(* Logix 5000 project; controller STAT 1756-L72 rev 20.12; software revision 20.04; part 8 of 34 *)
(* tags used below, declared in another part *)
   B14 : DINT[30];
   B3 : DINT[256];
   dmd_soude_ibt_ok : BOOL;
   FRANCK : BOOL;
   I10_000_Bit07 : ALIAS FOR I10[0].7;   // Hand Automaat CL8
   I10_001_Bit07 : ALIAS FOR I10[1].7;   // Hand Automaat CL9
   I19_000_Bit09 : ALIAS FOR I19[0].9;   // BP RESET KLAXON
   I1_008_Bit01 : ALIAS FOR I1[8].1;   // Hand Automaat stormbekken
   I8_001_Bit01 : ALIAS FOR I8[1].1;   // hand automaat cl5
   I8_001_Bit09 : ALIAS FOR I8[1].9;   // Schakelaar hand autom cl6
   I9_000_Bit09 : ALIAS FOR I9[0].9;   // Hand_Auto CL7
   ibt_level_soude_plein : BOOL;
   N12 : DINT[230];
   O12_000_Bit00 : ALIAS FOR O12[0].0;   // spoelpomp filters dubbele media P6_SPOEL
   O12_000_Bit01 : ALIAS FOR O12[0].1;   // pomp pompen uit kelder P23_KELDER
   O12_000_Bit02 : ALIAS FOR O12[0].2;   // pomp pompen uit kelder P24_KELDER
   O12_000_Bit03 : ALIAS FOR O12[0].3;   // motor ag1 mixer krimp neutralisatie AG1_MIXER_KRIMP
   O12_000_Bit08 : ALIAS FOR O12[0].8;   // pomp ag2 mixer vat 1 AG2_MIXER_VAT1
   O12_000_Bit09 : ALIAS FOR O12[0].9;   // pomp ag3 mixer vat 2 AG3_MIXER_VAT2
   O12_000_Bit10 : ALIAS FOR O12[0].10;   // pomp pd7 doseerpomp floculaat PD7_DOSEER_FLOCU
   O12_000_Bit11 : ALIAS FOR O12[0].11;   // pomp pd8 doseerpomp floculaat PD8_DOSEER_FLOCU
   O12_000_Bit12 : ALIAS FOR O12[0].12;   // Motor P19a zuiveringspomp controleweger P19_ZUIVERP
   O12_000_Bit13 : ALIAS FOR O12[0].13;   // Motor P20 zuiveringspomp controleweger P20_ZUIVERP
   O12_000_Bit14 : ALIAS FOR O12[0].14;   // Motor Pm1 recerculatiepomp ingang 1 decanter PM1_RECER_DEC1
   O12_000_Bit15 : ALIAS FOR O12[0].15;   // Motor Pm2 recerculatiepomp ingang 2 decanter PM2_RECER_DEC2
   O12_001_Bit00 : ALIAS FOR O12[1].0;   // Motor Pm3 evacuatiepomp ingang 1 decanter PM3_EVACU_IN_1
   O12_001_Bit01 : ALIAS FOR O12[1].1;   // Motor Pm4 evacuatiepomp ingang 2 decanter PM4_EVACU_IN_2
   O12_001_Bit03 : ALIAS FOR O12[1].3;   // Motor P7 voedingspomp omgekeerde osmose 1 P7_OSMOSE_1
   O12_001_Bit04 : ALIAS FOR O12[1].4;   // Motor P8 voedingspomp omgekeerde osmose 2 P8_OSMOSE_2
   O12_001_Bit05 : ALIAS FOR O12[1].5;   // Motor P9 voedingspomp omgekeerde osmose 3 P9_OSMOSE_3
   O14_001_Bit04 : ALIAS FOR O14[1].4;   // kalxon out NAOH
   O14_001_Bit05 : ALIAS FOR O14[1].5;   // lampe out NAOH
   O14_001_Bit06 : ALIAS FOR O14[1].6;   // klaxon out H2SO4
   O14_001_Bit07 : ALIAS FOR O14[1].7;   // lampe H2SO4
   O14_001_Bit08 : ALIAS FOR O14[1].8;   // klaxon out ZOUT
   O14_001_Bit09 : ALIAS FOR O14[1].9;   // lampe ZOUT
   O16_000_Bit09 : ALIAS FOR O16[0].9;   // LAMP_P17_AAN
   O16_000_Bit10 : ALIAS FOR O16[0].10;   // LAMP_P17_UIT
   O16_000_Bit11 : ALIAS FOR O16[0].11;   // LAMP_P18_AAN
   O16_000_Bit12 : ALIAS FOR O16[0].12;   // LAMP_P18_UIT
   O16_000_Bit15 : ALIAS FOR O16[0].15;   // LAMP_PRO1_AAN
   O16_001_Bit00 : ALIAS FOR O16[1].0;   // LAMP_PRO1_UIT
   O16_001_Bit01 : ALIAS FOR O16[1].1;   // LAMP_PRO2_AAN
   O16_001_Bit02 : ALIAS FOR O16[1].2;   // LAMP_PRO2_UIT
   O16_001_Bit03 : ALIAS FOR O16[1].3;   // LAMP_P21_AAN
   O16_001_Bit04 : ALIAS FOR O16[1].4;   // LAMP_P21_UIT
   O16_001_Bit05 : ALIAS FOR O16[1].5;   // LAMP_P22_AAN
   O16_001_Bit06 : ALIAS FOR O16[1].6;   // LAMP_P22_UIT
   O16_001_Bit07 : ALIAS FOR O16[1].7;   // LAMP_PRO3_AAN
   O16_001_Bit08 : ALIAS FOR O16[1].8;   // LAMP_PRO3_UIT
   O16_001_Bit09 : ALIAS FOR O16[1].9;   // LAMP_P21_REINIG_AAN
   O16_001_Bit10 : ALIAS FOR O16[1].10;   // LAMP_P21_REINIG_UIT
   O16_001_Bit11 : ALIAS FOR O16[1].11;   // LAMP_VENT_S1_AAN
   O16_001_Bit12 : ALIAS FOR O16[1].12;   // LAMP_VENT_S1_UIT
   O16_001_Bit13 : ALIAS FOR O16[1].13;   // LAMP_P3_AAN
   O16_001_Bit14 : ALIAS FOR O16[1].14;   // LAMP_P3_UIT
   O16_001_Bit15 : ALIAS FOR O16[1].15;   // LAMP_P4_AAN
   O17_000_Bit00 : ALIAS FOR O17[0].0;   // LAMP_P4_UIT
   O17_000_Bit01 : ALIAS FOR O17[0].1;   // LAMP_P5_AAN
   O17_000_Bit02 : ALIAS FOR O17[0].2;   // LAMP_P5_UIT
   O17_000_Bit03 : ALIAS FOR O17[0].3;   // LAMP_P6_AAN
   O17_000_Bit04 : ALIAS FOR O17[0].4;   // LAMP_P6_UIT
   O17_000_Bit05 : ALIAS FOR O17[0].5;   // LAMP_P23_AAN
   O17_000_Bit06 : ALIAS FOR O17[0].6;   // LAMP_P23_UIT
   O17_000_Bit07 : ALIAS FOR O17[0].7;   // LAMP_P24_AAN
   O17_000_Bit08 : ALIAS FOR O17[0].8;   // LAMP_P24_UIT
   O17_000_Bit09 : ALIAS FOR O17[0].9;   // LAMP_AG1_AAN
   O17_000_Bit10 : ALIAS FOR O17[0].10;   // LAMP_AG1_UIT
   O17_000_Bit11 : ALIAS FOR O17[0].11;   // LAMP_AG2_AAN
   O17_000_Bit12 : ALIAS FOR O17[0].12;   // LAMP_AG2_UIT
   O17_000_Bit13 : ALIAS FOR O17[0].13;   // LAMP_AG3_AAN
   O17_000_Bit14 : ALIAS FOR O17[0].14;   // LAMP_AG3_UIT
   O17_000_Bit15 : ALIAS FOR O17[0].15;   // LAMP_PD7_AAN
   O17_001_Bit00 : ALIAS FOR O17[1].0;   // LAMP_PD7_UIT
   O17_001_Bit01 : ALIAS FOR O17[1].1;   // LAMP_PD8_AAN
   O17_001_Bit02 : ALIAS FOR O17[1].2;   // LAMP_PD8_UIT
   O17_001_Bit03 : ALIAS FOR O17[1].3;   // LAMP_P19A_AAN
   O17_001_Bit04 : ALIAS FOR O17[1].4;   // LAMP_P19A_UIT
   O17_001_Bit05 : ALIAS FOR O17[1].5;   // LAMP_P19B_AAN
   O17_001_Bit06 : ALIAS FOR O17[1].6;   // LAMP_P19B_UIT
   O17_001_Bit09 : ALIAS FOR O17[1].9;   // LAMP_P25_AAN
   O17_001_Bit10 : ALIAS FOR O17[1].10;   // LAMP_P25_UIT
   O17_001_Bit11 : ALIAS FOR O17[1].11;   // LAMP_PM1_AAN
   O17_001_Bit12 : ALIAS FOR O17[1].12;   // LAMP_PM1_UIT
   O17_001_Bit13 : ALIAS FOR O17[1].13;   // LAMP_PM2_AAN
   O17_001_Bit14 : ALIAS FOR O17[1].14;   // LAMP_PM2_UIT
   O17_001_Bit15 : ALIAS FOR O17[1].15;   // LAMP_PM3_AAN
   O18_000_Bit00 : ALIAS FOR O18[0].0;   // LAMP_PM3_UIT
   O18_000_Bit01 : ALIAS FOR O18[0].1;   // LAMP_PM4_AAN
   O18_000_Bit02 : ALIAS FOR O18[0].2;   // LAMP_PM4_UIT
   O18_000_Bit07 : ALIAS FOR O18[0].7;   // LAMP_P7_AAN
   O18_000_Bit08 : ALIAS FOR O18[0].8;   // LAMP_P7_UIT
   O18_000_Bit09 : ALIAS FOR O18[0].9;   // LAMP_P8_AAN
   O18_000_Bit10 : ALIAS FOR O18[0].10;   // LAMP_P8_UIT
   O18_000_Bit11 : ALIAS FOR O18[0].11;   // LAMP_P9_AAN
   O18_000_Bit12 : ALIAS FOR O18[0].12;   // LAMP_P9_UIT
   O1_006_Bit15 : ALIAS FOR O1[6].15;
   O1_011_Bit00 : ALIAS FOR O1[11].0;
   O1_011_Bit03 : ALIAS FOR O1[11].3;
   O1_011_Bit06 : ALIAS FOR O1[11].6;
   O1_011_Bit09 : ALIAS FOR O1[11].9;
   O1_011_Bit10 : ALIAS FOR O1[11].10;
   O1_012_Bit01 : ALIAS FOR O1[12].1;
   O1_012_Bit02 : ALIAS FOR O1[12].2;
   O1_012_Bit03 : ALIAS FOR O1[12].3;
   O1_012_Bit04 : ALIAS FOR O1[12].4;
   O1_012_Bit05 : ALIAS FOR O1[12].5;
   O1_012_Bit06 : ALIAS FOR O1[12].6;
   O1_012_Bit07 : ALIAS FOR O1[12].7;
   O1_012_Bit08 : ALIAS FOR O1[12].8;
   O1_012_Bit09 : ALIAS FOR O1[12].9;
   O1_012_Bit10 : ALIAS FOR O1[12].10;
   s_bp_stop_soude_ibt : BOOL;
   S_dmd_naoh_ibt : REAL;
   S_naoh_ibt_passe : REAL;
   soude_ibt_fini : BOOL;
   T1_cligno : TIMER;
   T2_cligno : TIMER;

PROGRAM ibt   (* main routine ibtmain *)
VAR
   INT0 : INT := 6;
   INT1 : INT := -21846;
   P21 : BOOL;
   P22 : BOOL;
END_VAR

ROUTINE _10_LAMPES   (* ladder *)
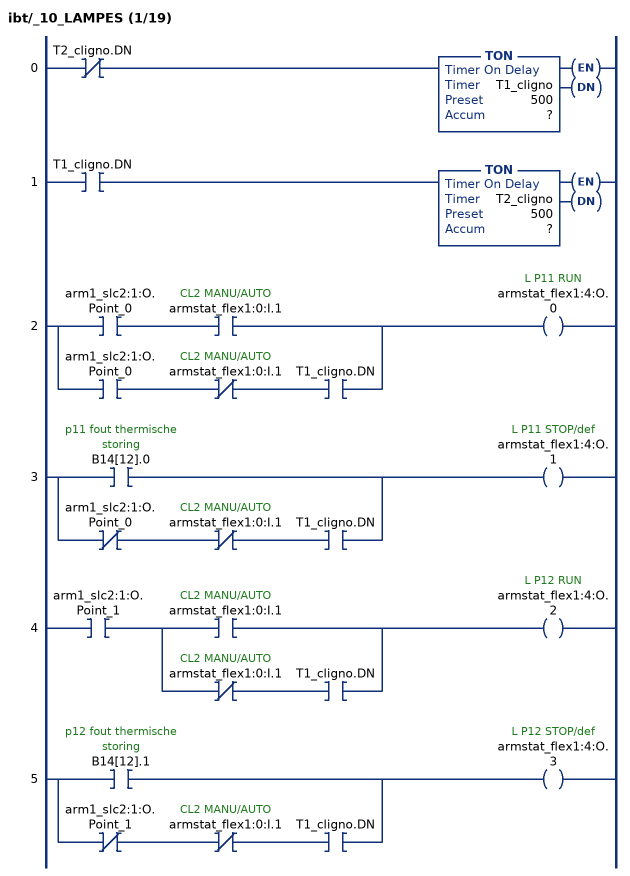
   0: XIO(T2_cligno.DN)TON(T1_cligno,?,?);
   1: XIC(T1_cligno.DN)TON(T2_cligno,?,?);
   2: [XIC(arm1_slc2:1:O.Point_0) XIC(armstat_flex1:0:I.1) ,XIC(arm1_slc2:1:O.Point_0) XIO(armstat_flex1:0:I.1) XIC(T1_cligno.DN) ]OTE(armstat_flex1:4:O.0);
   3: [XIC(B14[12].0) ,XIO(arm1_slc2:1:O.Point_0) XIO(armstat_flex1:0:I.1) XIC(T1_cligno.DN) ]OTE(armstat_flex1:4:O.1);
   4: XIC(arm1_slc2:1:O.Point_1)[XIC(armstat_flex1:0:I.1) ,XIO(armstat_flex1:0:I.1) XIC(T1_cligno.DN) ]OTE(armstat_flex1:4:O.2);
   5: [XIC(B14[12].1) ,XIO(arm1_slc2:1:O.Point_1) XIO(armstat_flex1:0:I.1) XIC(T1_cligno.DN) ]OTE(armstat_flex1:4:O.3);
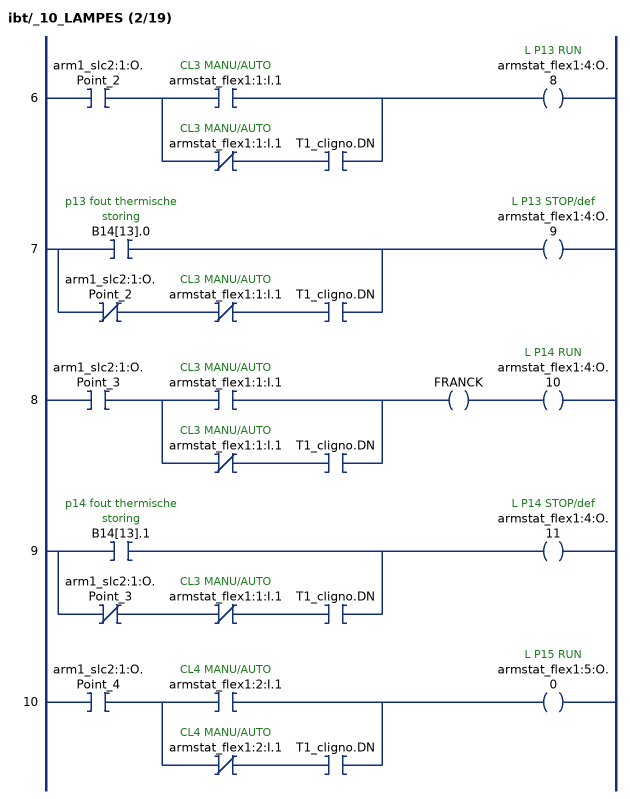
   6: XIC(arm1_slc2:1:O.Point_2)[XIC(armstat_flex1:1:I.1) ,XIO(armstat_flex1:1:I.1) XIC(T1_cligno.DN) ]OTE(armstat_flex1:4:O.8);
   7: [XIC(B14[13].0) ,XIO(arm1_slc2:1:O.Point_2) XIO(armstat_flex1:1:I.1) XIC(T1_cligno.DN) ]OTE(armstat_flex1:4:O.9);
   8: XIC(arm1_slc2:1:O.Point_3)[XIC(armstat_flex1:1:I.1) ,XIO(armstat_flex1:1:I.1) XIC(T1_cligno.DN) ]OTE(FRANCK)OTE(armstat_flex1:4:O.10);
   9: [XIC(B14[13].1) ,XIO(arm1_slc2:1:O.Point_3) XIO(armstat_flex1:1:I.1) XIC(T1_cligno.DN) ]OTE(armstat_flex1:4:O.11);
   10: XIC(arm1_slc2:1:O.Point_4)[XIC(armstat_flex1:2:I.1) ,XIO(armstat_flex1:2:I.1) XIC(T1_cligno.DN) ]OTE(armstat_flex1:5:O.0);
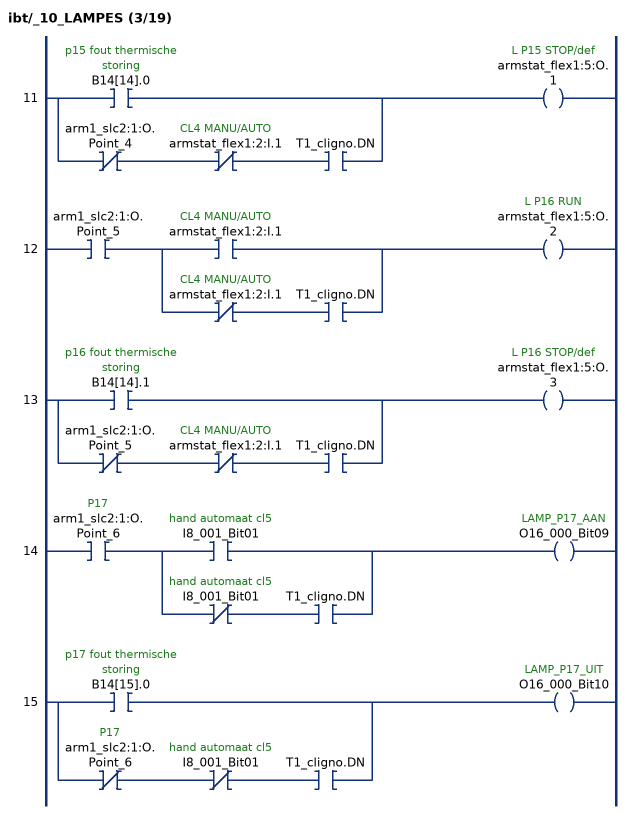
   11: [XIC(B14[14].0) ,XIO(arm1_slc2:1:O.Point_4) XIO(armstat_flex1:2:I.1) XIC(T1_cligno.DN) ]OTE(armstat_flex1:5:O.1);
   12: XIC(arm1_slc2:1:O.Point_5)[XIC(armstat_flex1:2:I.1) ,XIO(armstat_flex1:2:I.1) XIC(T1_cligno.DN) ]OTE(armstat_flex1:5:O.2);
   13: [XIC(B14[14].1) ,XIO(arm1_slc2:1:O.Point_5) XIO(armstat_flex1:2:I.1) XIC(T1_cligno.DN) ]OTE(armstat_flex1:5:O.3);
   14: XIC(arm1_slc2:1:O.Point_6)[XIC(I8_001_Bit01) ,XIO(I8_001_Bit01) XIC(T1_cligno.DN) ]OTE(O16_000_Bit09);
   15: [XIC(B14[15].0) ,XIO(arm1_slc2:1:O.Point_6) XIO(I8_001_Bit01) XIC(T1_cligno.DN) ]OTE(O16_000_Bit10);
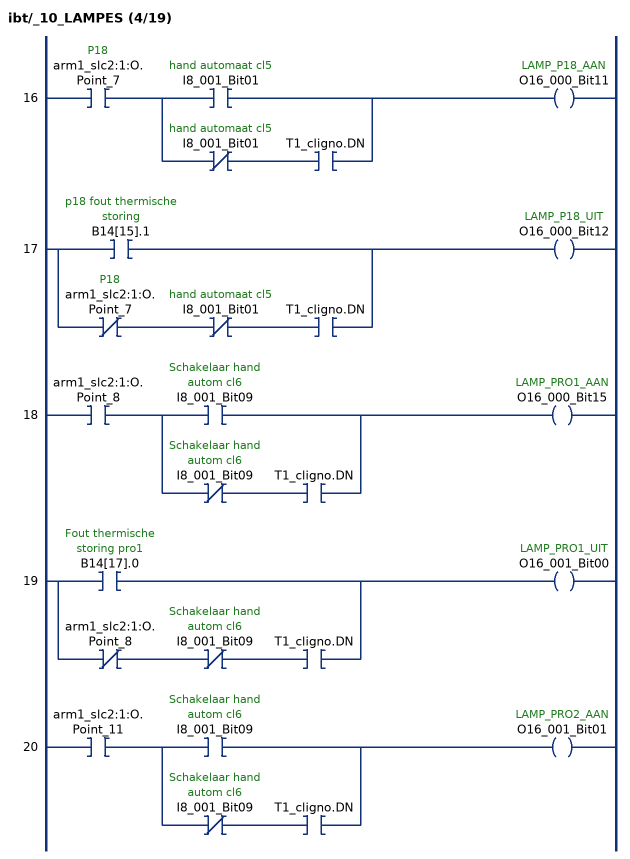
   16: XIC(arm1_slc2:1:O.Point_7)[XIC(I8_001_Bit01) ,XIO(I8_001_Bit01) XIC(T1_cligno.DN) ]OTE(O16_000_Bit11);
   17: [XIC(B14[15].1) ,XIO(arm1_slc2:1:O.Point_7) XIO(I8_001_Bit01) XIC(T1_cligno.DN) ]OTE(O16_000_Bit12);
   18: XIC(arm1_slc2:1:O.Point_8)[XIC(I8_001_Bit09) ,XIO(I8_001_Bit09) XIC(T1_cligno.DN) ]OTE(O16_000_Bit15);
   19: [XIC(B14[17].0) ,XIO(arm1_slc2:1:O.Point_8) XIO(I8_001_Bit09) XIC(T1_cligno.DN) ]OTE(O16_001_Bit00);
   20: XIC(arm1_slc2:1:O.Point_11)[XIC(I8_001_Bit09) ,XIO(I8_001_Bit09) XIC(T1_cligno.DN) ]OTE(O16_001_Bit01);
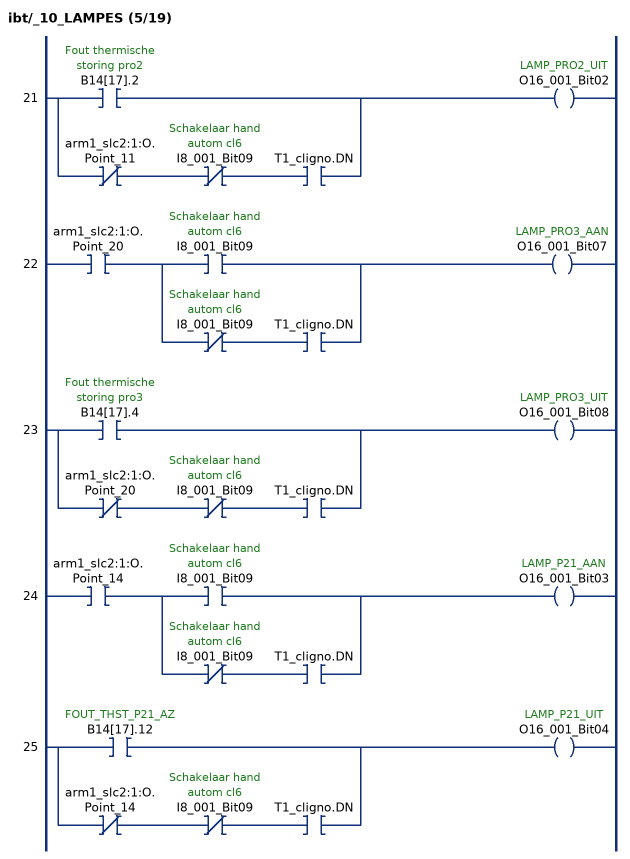
   21: [XIC(B14[17].2) ,XIO(arm1_slc2:1:O.Point_11) XIO(I8_001_Bit09) XIC(T1_cligno.DN) ]OTE(O16_001_Bit02);
   22: XIC(arm1_slc2:1:O.Point_20)[XIC(I8_001_Bit09) ,XIO(I8_001_Bit09) XIC(T1_cligno.DN) ]OTE(O16_001_Bit07);
   23: [XIC(B14[17].4) ,XIO(arm1_slc2:1:O.Point_20) XIO(I8_001_Bit09) XIC(T1_cligno.DN) ]OTE(O16_001_Bit08);
   24: XIC(arm1_slc2:1:O.Point_14)[XIC(I8_001_Bit09) ,XIO(I8_001_Bit09) XIC(T1_cligno.DN) ]OTE(O16_001_Bit03);
   25: [XIC(B14[17].12) ,XIO(arm1_slc2:1:O.Point_14) XIO(I8_001_Bit09) XIC(T1_cligno.DN) ]OTE(O16_001_Bit04);
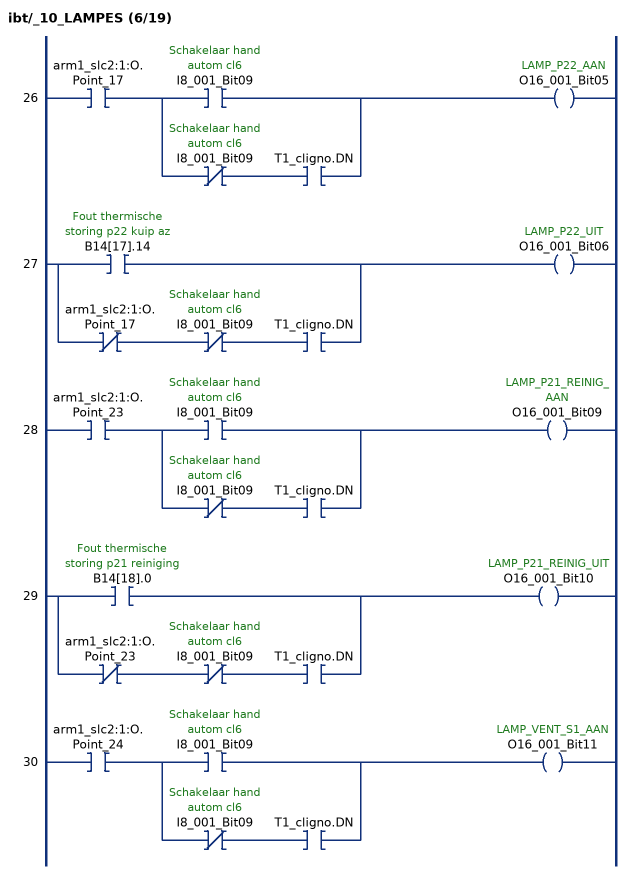
   26: XIC(arm1_slc2:1:O.Point_17)[XIC(I8_001_Bit09) ,XIO(I8_001_Bit09) XIC(T1_cligno.DN) ]OTE(O16_001_Bit05);
   27: [XIC(B14[17].14) ,XIO(arm1_slc2:1:O.Point_17) XIO(I8_001_Bit09) XIC(T1_cligno.DN) ]OTE(O16_001_Bit06);
   28: XIC(arm1_slc2:1:O.Point_23)[XIC(I8_001_Bit09) ,XIO(I8_001_Bit09) XIC(T1_cligno.DN) ]OTE(O16_001_Bit09);
   29: [XIC(B14[18].0) ,XIO(arm1_slc2:1:O.Point_23) XIO(I8_001_Bit09) XIC(T1_cligno.DN) ]OTE(O16_001_Bit10);
   30: XIC(arm1_slc2:1:O.Point_24)[XIC(I8_001_Bit09) ,XIO(I8_001_Bit09) XIC(T1_cligno.DN) ]OTE(O16_001_Bit11);
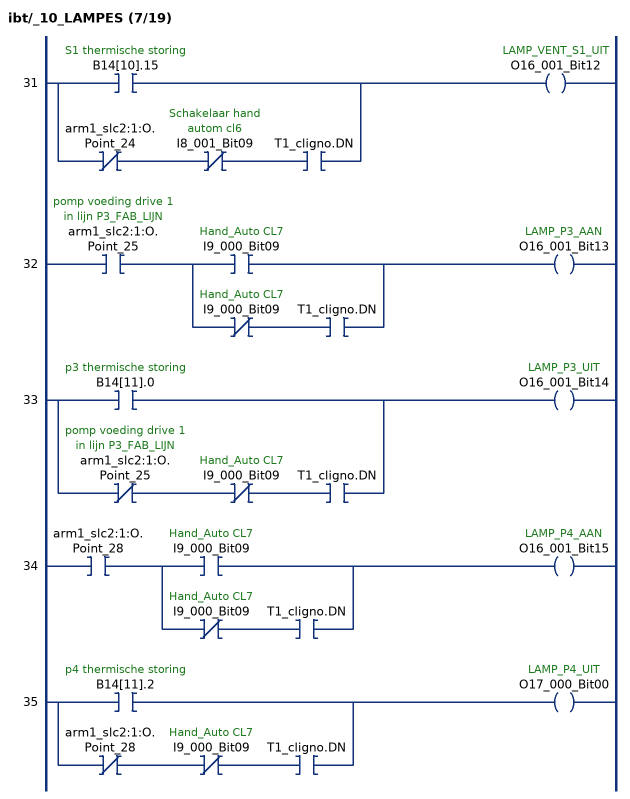
   31: [XIC(B14[10].15) ,XIO(arm1_slc2:1:O.Point_24) XIO(I8_001_Bit09) XIC(T1_cligno.DN) ]OTE(O16_001_Bit12);
   32: XIC(arm1_slc2:1:O.Point_25)[XIC(I9_000_Bit09) ,XIO(I9_000_Bit09) XIC(T1_cligno.DN) ]OTE(O16_001_Bit13);
   33: [XIC(B14[11].0) ,XIO(arm1_slc2:1:O.Point_25) XIO(I9_000_Bit09) XIC(T1_cligno.DN) ]OTE(O16_001_Bit14);
   34: XIC(arm1_slc2:1:O.Point_28)[XIC(I9_000_Bit09) ,XIO(I9_000_Bit09) XIC(T1_cligno.DN) ]OTE(O16_001_Bit15);
   35: [XIC(B14[11].2) ,XIO(arm1_slc2:1:O.Point_28) XIO(I9_000_Bit09) XIC(T1_cligno.DN) ]OTE(O17_000_Bit00);
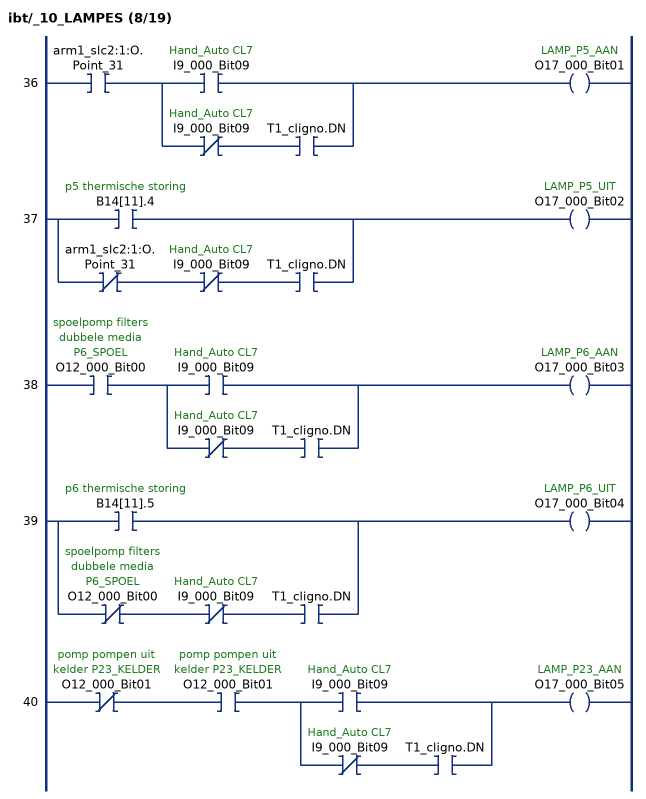
   36: XIC(arm1_slc2:1:O.Point_31)[XIC(I9_000_Bit09) ,XIO(I9_000_Bit09) XIC(T1_cligno.DN) ]OTE(O17_000_Bit01);
   37: [XIC(B14[11].4) ,XIO(arm1_slc2:1:O.Point_31) XIO(I9_000_Bit09) XIC(T1_cligno.DN) ]OTE(O17_000_Bit02);
   38: XIC(O12_000_Bit00)[XIC(I9_000_Bit09) ,XIO(I9_000_Bit09) XIC(T1_cligno.DN) ]OTE(O17_000_Bit03);
   39: [XIC(B14[11].5) ,XIO(O12_000_Bit00) XIO(I9_000_Bit09) XIC(T1_cligno.DN) ]OTE(O17_000_Bit04);
   40: XIO(O12_000_Bit01)XIC(O12_000_Bit01)[XIC(I9_000_Bit09) ,XIO(I9_000_Bit09) XIC(T1_cligno.DN) ]OTE(O17_000_Bit05);
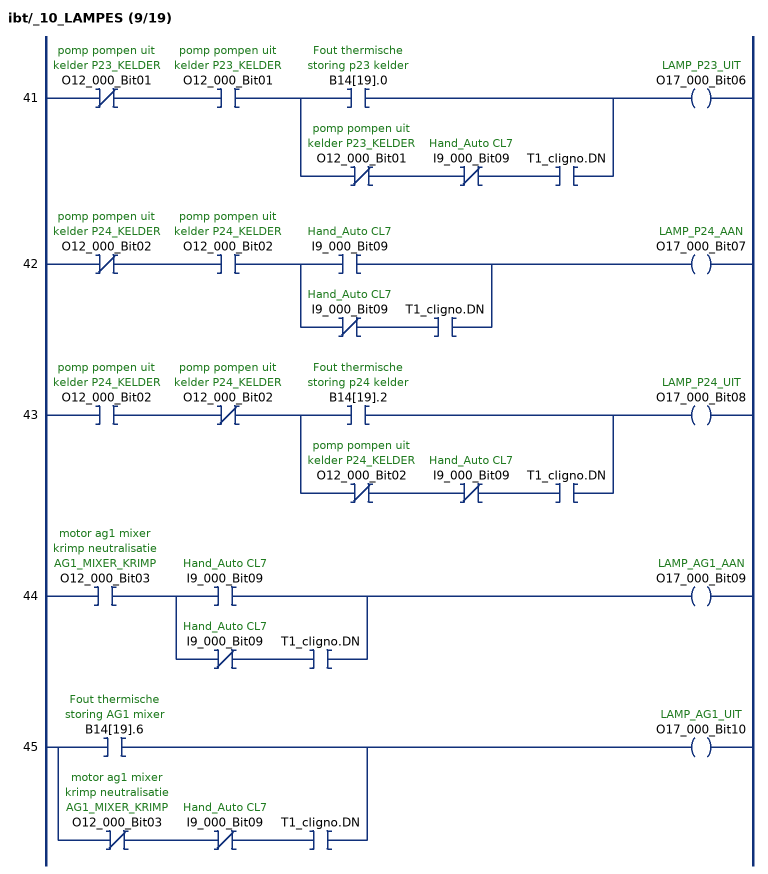
   41: XIO(O12_000_Bit01)XIC(O12_000_Bit01)[XIC(B14[19].0) ,XIO(O12_000_Bit01) XIO(I9_000_Bit09) XIC(T1_cligno.DN) ]OTE(O17_000_Bit06);
   42: XIO(O12_000_Bit02)XIC(O12_000_Bit02)[XIC(I9_000_Bit09) ,XIO(I9_000_Bit09) XIC(T1_cligno.DN) ]OTE(O17_000_Bit07);
   43: XIC(O12_000_Bit02)XIO(O12_000_Bit02)[XIC(B14[19].2) ,XIO(O12_000_Bit02) XIO(I9_000_Bit09) XIC(T1_cligno.DN) ]OTE(O17_000_Bit08);
   44: XIC(O12_000_Bit03)[XIC(I9_000_Bit09) ,XIO(I9_000_Bit09) XIC(T1_cligno.DN) ]OTE(O17_000_Bit09);
   45: [XIC(B14[19].6) ,XIO(O12_000_Bit03) XIO(I9_000_Bit09) XIC(T1_cligno.DN) ]OTE(O17_000_Bit10);
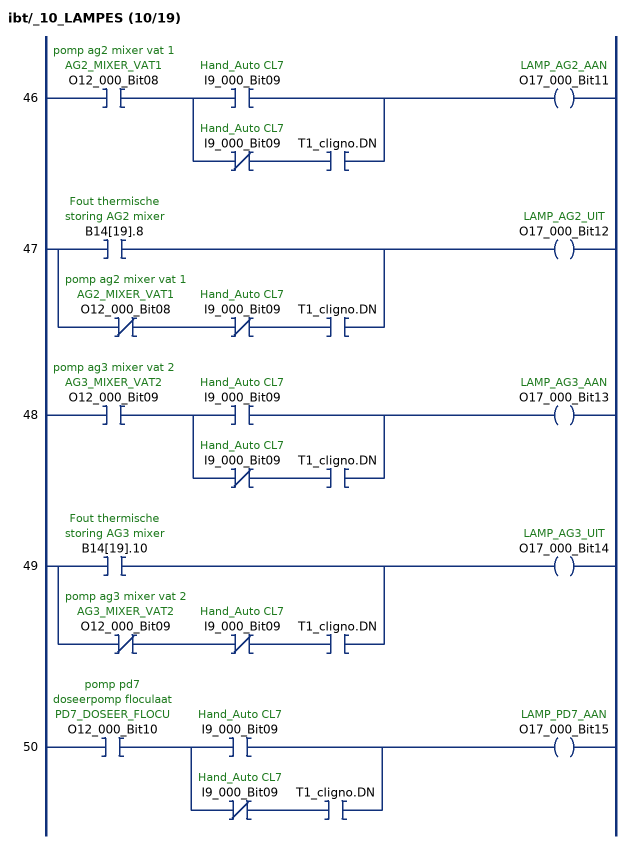
   46: XIC(O12_000_Bit08)[XIC(I9_000_Bit09) ,XIO(I9_000_Bit09) XIC(T1_cligno.DN) ]OTE(O17_000_Bit11);
   47: [XIC(B14[19].8) ,XIO(O12_000_Bit08) XIO(I9_000_Bit09) XIC(T1_cligno.DN) ]OTE(O17_000_Bit12);
   48: XIC(O12_000_Bit09)[XIC(I9_000_Bit09) ,XIO(I9_000_Bit09) XIC(T1_cligno.DN) ]OTE(O17_000_Bit13);
   49: [XIC(B14[19].10) ,XIO(O12_000_Bit09) XIO(I9_000_Bit09) XIC(T1_cligno.DN) ]OTE(O17_000_Bit14);
   50: XIC(O12_000_Bit10)[XIC(I9_000_Bit09) ,XIO(I9_000_Bit09) XIC(T1_cligno.DN) ]OTE(O17_000_Bit15);
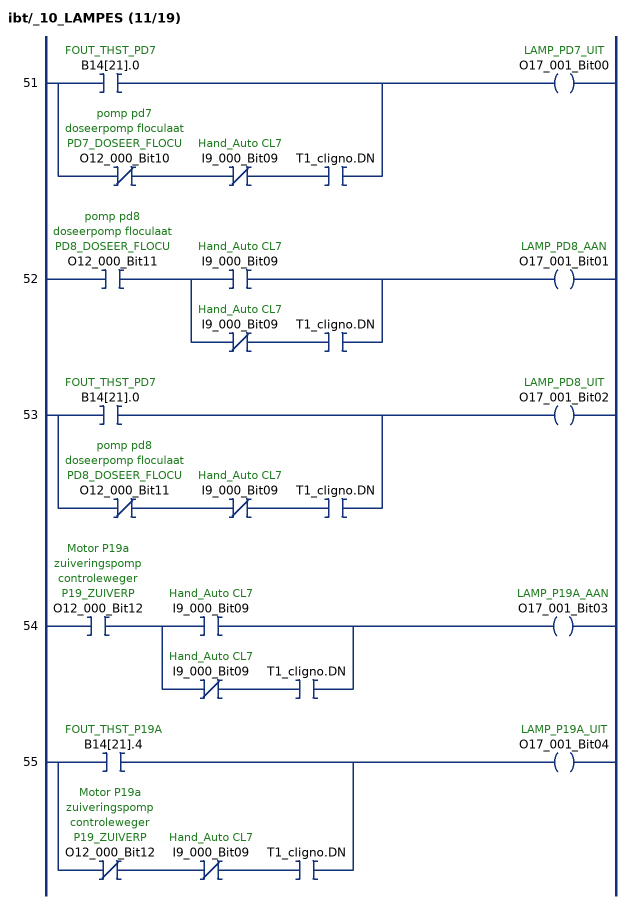
   51: [XIC(B14[21].0) ,XIO(O12_000_Bit10) XIO(I9_000_Bit09) XIC(T1_cligno.DN) ]OTE(O17_001_Bit00);
   52: XIC(O12_000_Bit11)[XIC(I9_000_Bit09) ,XIO(I9_000_Bit09) XIC(T1_cligno.DN) ]OTE(O17_001_Bit01);
   53: [XIC(B14[21].0) ,XIO(O12_000_Bit11) XIO(I9_000_Bit09) XIC(T1_cligno.DN) ]OTE(O17_001_Bit02);
   54: XIC(O12_000_Bit12)[XIC(I9_000_Bit09) ,XIO(I9_000_Bit09) XIC(T1_cligno.DN) ]OTE(O17_001_Bit03);
   55: [XIC(B14[21].4) ,XIO(O12_000_Bit12) XIO(I9_000_Bit09) XIC(T1_cligno.DN) ]OTE(O17_001_Bit04);
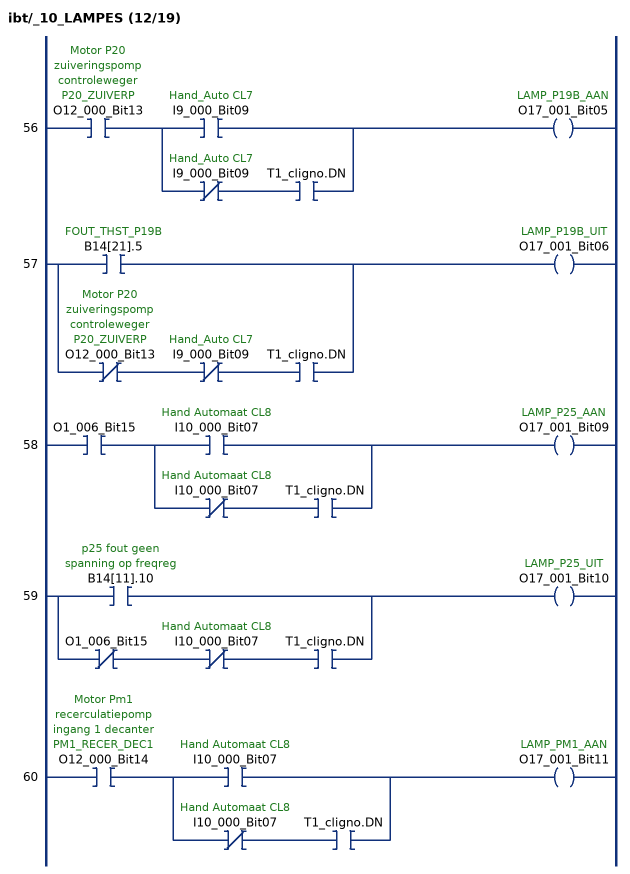
   56: XIC(O12_000_Bit13)[XIC(I9_000_Bit09) ,XIO(I9_000_Bit09) XIC(T1_cligno.DN) ]OTE(O17_001_Bit05);
   57: [XIC(B14[21].5) ,XIO(O12_000_Bit13) XIO(I9_000_Bit09) XIC(T1_cligno.DN) ]OTE(O17_001_Bit06);
   58: XIC(O1_006_Bit15)[XIC(I10_000_Bit07) ,XIO(I10_000_Bit07) XIC(T1_cligno.DN) ]OTE(O17_001_Bit09);
   59: [XIC(B14[11].10) ,XIO(O1_006_Bit15) XIO(I10_000_Bit07) XIC(T1_cligno.DN) ]OTE(O17_001_Bit10);
   60: XIC(O12_000_Bit14)[XIC(I10_000_Bit07) ,XIO(I10_000_Bit07) XIC(T1_cligno.DN) ]OTE(O17_001_Bit11);
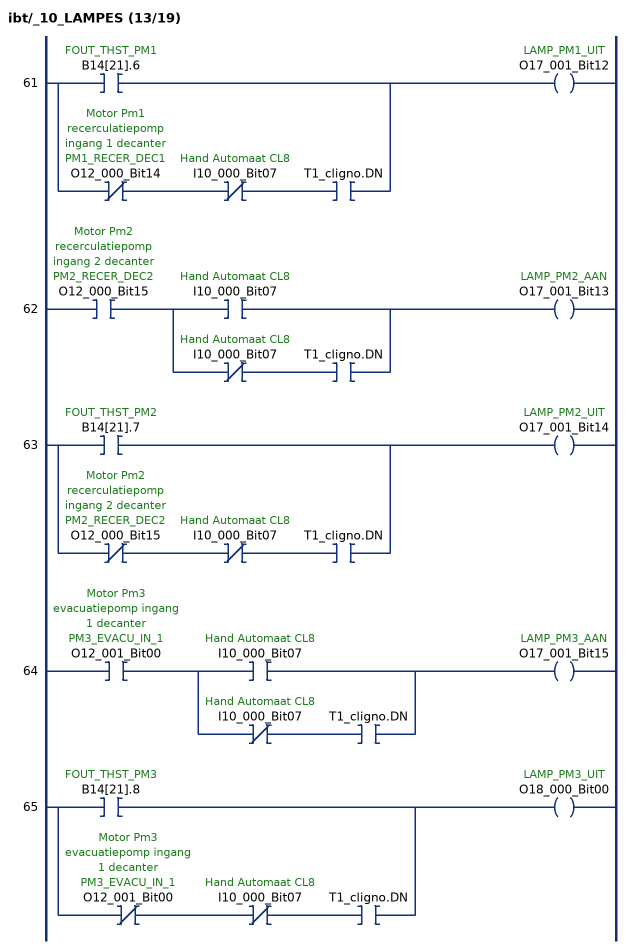
   61: [XIC(B14[21].6) ,XIO(O12_000_Bit14) XIO(I10_000_Bit07) XIC(T1_cligno.DN) ]OTE(O17_001_Bit12);
   62: XIC(O12_000_Bit15)[XIC(I10_000_Bit07) ,XIO(I10_000_Bit07) XIC(T1_cligno.DN) ]OTE(O17_001_Bit13);
   63: [XIC(B14[21].7) ,XIO(O12_000_Bit15) XIO(I10_000_Bit07) XIC(T1_cligno.DN) ]OTE(O17_001_Bit14);
   64: XIC(O12_001_Bit00)[XIC(I10_000_Bit07) ,XIO(I10_000_Bit07) XIC(T1_cligno.DN) ]OTE(O17_001_Bit15);
   65: [XIC(B14[21].8) ,XIO(O12_001_Bit00) XIO(I10_000_Bit07) XIC(T1_cligno.DN) ]OTE(O18_000_Bit00);
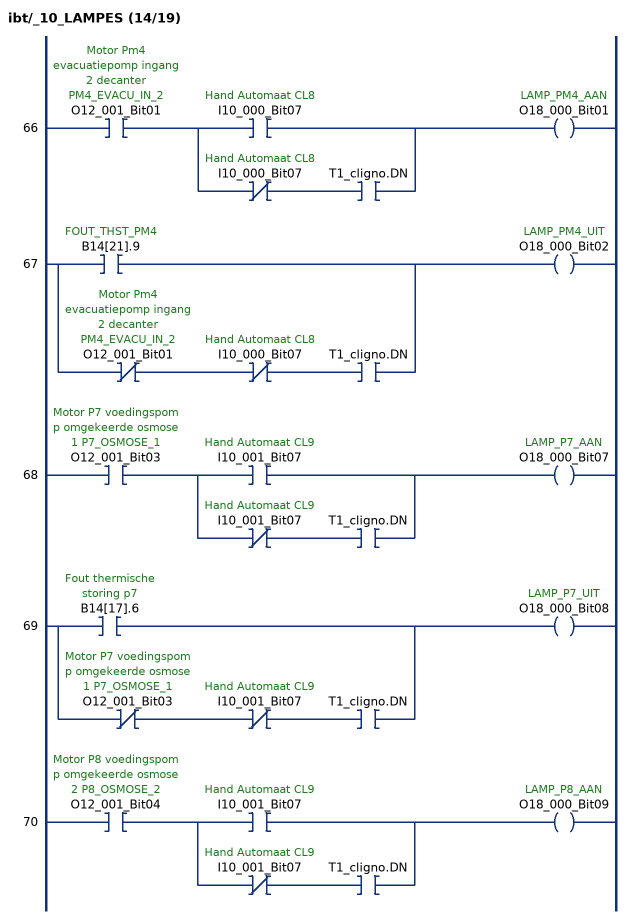
   66: XIC(O12_001_Bit01)[XIC(I10_000_Bit07) ,XIO(I10_000_Bit07) XIC(T1_cligno.DN) ]OTE(O18_000_Bit01);
   67: [XIC(B14[21].9) ,XIO(O12_001_Bit01) XIO(I10_000_Bit07) XIC(T1_cligno.DN) ]OTE(O18_000_Bit02);
   68: XIC(O12_001_Bit03)[XIC(I10_001_Bit07) ,XIO(I10_001_Bit07) XIC(T1_cligno.DN) ]OTE(O18_000_Bit07);
   69: [XIC(B14[17].6) ,XIO(O12_001_Bit03) XIO(I10_001_Bit07) XIC(T1_cligno.DN) ]OTE(O18_000_Bit08);
   70: XIC(O12_001_Bit04)[XIC(I10_001_Bit07) ,XIO(I10_001_Bit07) XIC(T1_cligno.DN) ]OTE(O18_000_Bit09);
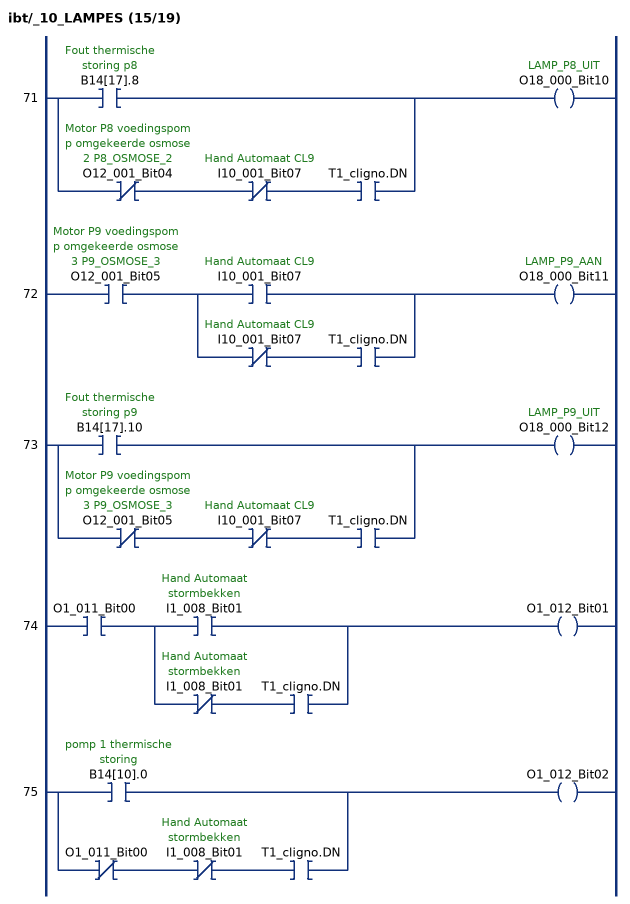
   71: [XIC(B14[17].8) ,XIO(O12_001_Bit04) XIO(I10_001_Bit07) XIC(T1_cligno.DN) ]OTE(O18_000_Bit10);
   72: XIC(O12_001_Bit05)[XIC(I10_001_Bit07) ,XIO(I10_001_Bit07) XIC(T1_cligno.DN) ]OTE(O18_000_Bit11);
   73: [XIC(B14[17].10) ,XIO(O12_001_Bit05) XIO(I10_001_Bit07) XIC(T1_cligno.DN) ]OTE(O18_000_Bit12);
   74: XIC(O1_011_Bit00)[XIC(I1_008_Bit01) ,XIO(I1_008_Bit01) XIC(T1_cligno.DN) ]OTE(O1_012_Bit01);
   75: [XIC(B14[10].0) ,XIO(O1_011_Bit00) XIO(I1_008_Bit01) XIC(T1_cligno.DN) ]OTE(O1_012_Bit02);
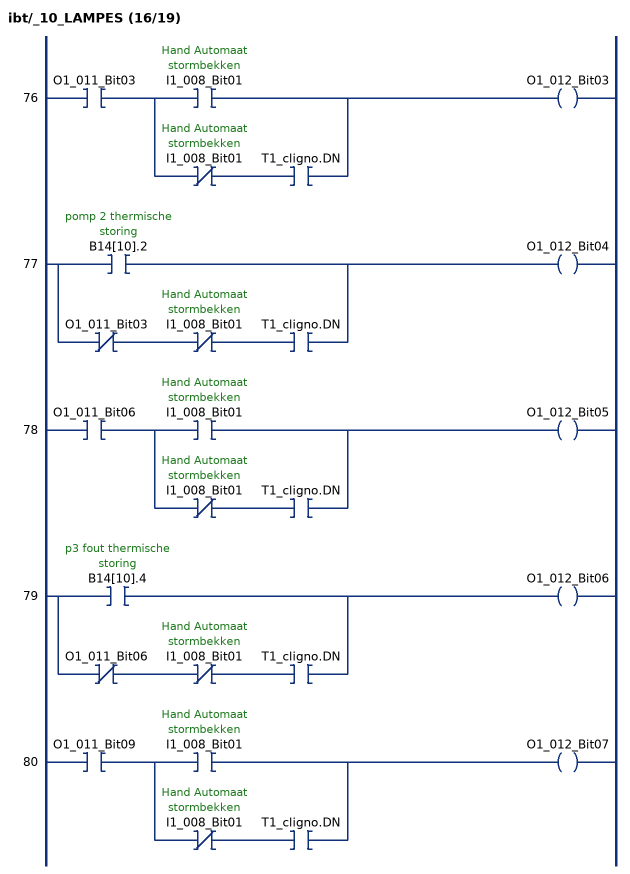
   76: XIC(O1_011_Bit03)[XIC(I1_008_Bit01) ,XIO(I1_008_Bit01) XIC(T1_cligno.DN) ]OTE(O1_012_Bit03);
   77: [XIC(B14[10].2) ,XIO(O1_011_Bit03) XIO(I1_008_Bit01) XIC(T1_cligno.DN) ]OTE(O1_012_Bit04);
   78: XIC(O1_011_Bit06)[XIC(I1_008_Bit01) ,XIO(I1_008_Bit01) XIC(T1_cligno.DN) ]OTE(O1_012_Bit05);
   79: [XIC(B14[10].4) ,XIO(O1_011_Bit06) XIO(I1_008_Bit01) XIC(T1_cligno.DN) ]OTE(O1_012_Bit06);
   80: XIC(O1_011_Bit09)[XIC(I1_008_Bit01) ,XIO(I1_008_Bit01) XIC(T1_cligno.DN) ]OTE(O1_012_Bit07);
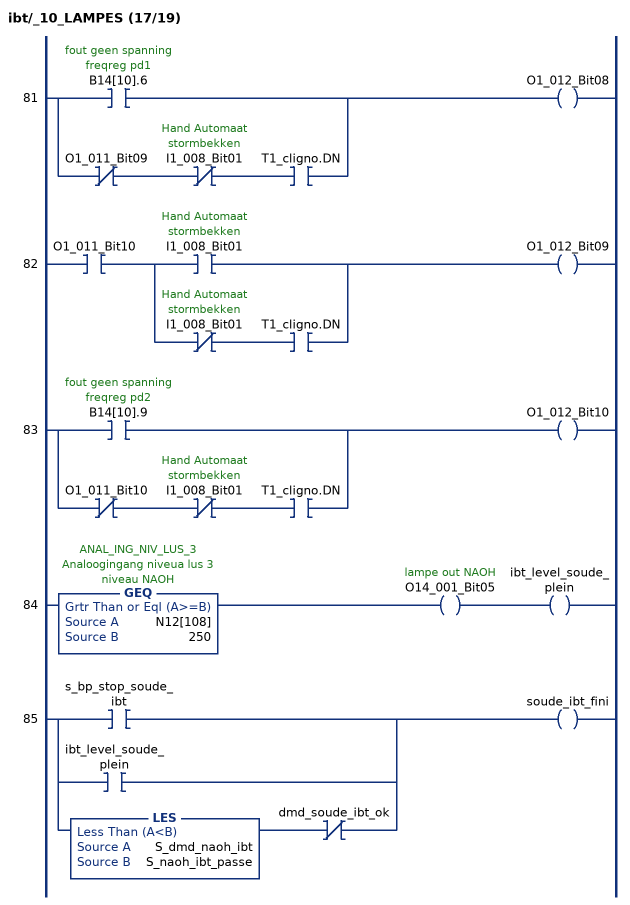
   81: [XIC(B14[10].6) ,XIO(O1_011_Bit09) XIO(I1_008_Bit01) XIC(T1_cligno.DN) ]OTE(O1_012_Bit08);
   82: XIC(O1_011_Bit10)[XIC(I1_008_Bit01) ,XIO(I1_008_Bit01) XIC(T1_cligno.DN) ]OTE(O1_012_Bit09);
   83: [XIC(B14[10].9) ,XIO(O1_011_Bit10) XIO(I1_008_Bit01) XIC(T1_cligno.DN) ]OTE(O1_012_Bit10);
   84: GEQ(N12[108],250)OTE(O14_001_Bit05)OTE(ibt_level_soude_plein);
   85: [XIC(s_bp_stop_soude_ibt) ,XIC(ibt_level_soude_plein) ,LES(S_dmd_naoh_ibt,S_naoh_ibt_passe) XIO(dmd_soude_ibt_ok) ]OTE(soude_ibt_fini);
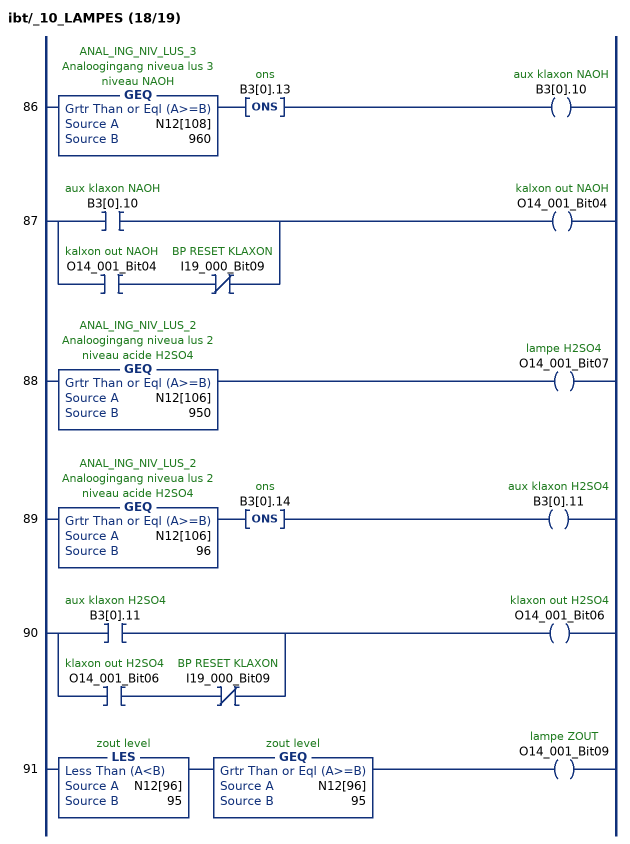
   86: GEQ(N12[108],960)ONS(B3[0].13)OTE(B3[0].10);
   87: [XIC(B3[0].10) ,XIC(O14_001_Bit04) XIO(I19_000_Bit09) ]OTE(O14_001_Bit04);
   88: GEQ(N12[106],950)OTE(O14_001_Bit07);
   89: GEQ(N12[106],96)ONS(B3[0].14)OTE(B3[0].11);
   90: [XIC(B3[0].11) ,XIC(O14_001_Bit06) XIO(I19_000_Bit09) ]OTE(O14_001_Bit06);
   91: LES(N12[96],95)GEQ(N12[96],95)OTE(O14_001_Bit09);
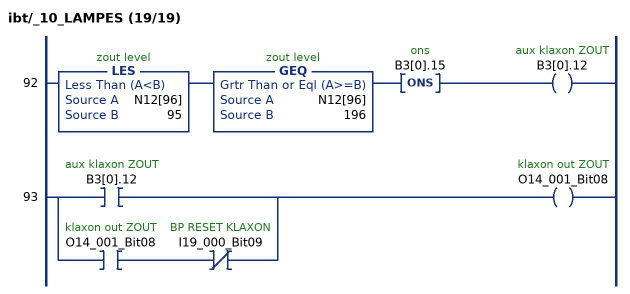
   92: LES(N12[96],95)GEQ(N12[96],196)ONS(B3[0].15)OTE(B3[0].12);
   93: [XIC(B3[0].12) ,XIC(O14_001_Bit08) XIO(I19_000_Bit09) ]OTE(O14_001_Bit08);
END_ROUTINE
